// TIA Portal V20 export
DATA_BLOCK "HMI_SideShifter_1"   // DB2
{ S7_Optimized_Access := 'TRUE' }
// stored: MemoryReserve 100
   VAR
      SL_Go_Forward : Bool;
      SL_Go_Backward : Bool;
      SL_Velocity : Int;
      SL_Hydraulic_Unit : Bool;
      SL_Actuators_Push : Bool;
      SL_Actuators_Pull : Bool;
      Go_to_ST35 : Bool;
      Go_to_ST02 : Bool;
      Go_to_ST03 : Bool;
      Go_to_ST04 : Bool;
      SR_SL_Hyd_Up : Bool;
      SR_SL_Hyd_Down : Bool;
      SR_Go_Forward : Bool;
      SR_Go_Backward : Bool;
      SR_Velocity : Int;
      SR_Hydraulic_Unit : Bool;
      SR_Actuators_Push : Bool;
      SR_Actuators_Pull : Bool;
      Reset_Drives : Bool;
      Reset_Hydro : Bool;
   END_VAR
   VAR RETAIN
      Homing_SL1 { S7_SetPoint := 'True'} : Int := 1850;
      Homing_SL2 { S7_SetPoint := 'True'} : Int := 7446;
      Homing_SL3 { S7_SetPoint := 'True'} : Int := 13443;
      Homing_SL4 { S7_SetPoint := 'True'} : Int := 19050;
      Homing_SR1 { S7_SetPoint := 'True'} : Int := 1853;
      Homing_SR2 { S7_SetPoint := 'True'} : Int := 7449;
      Homing_SR3 { S7_SetPoint := 'True'} : Int := 13454;
      Homing_SR4 { S7_SetPoint := 'True'} : Int := 19050;
   END_VAR
BEGIN
END_DATA_BLOCK
